(* PLC project SafeLOGIC-1, BrAutomation SafeDESIGNER  4.1.3.320 *)
(* stored: companyURL http://www.br-automation.com, creationDateTime Thu May 07 13:59:02 2020 *)

PROGRAM Zone
  VAR  (* added by the conversion: wires and edge detectors of the diagram *)
    _SAFEBOOL_TO_BOOL91_OUT : BOOL;
    _BOOL_TO_SAFEBOOL159_OUT : SAFEBOOL;
  END_VAR

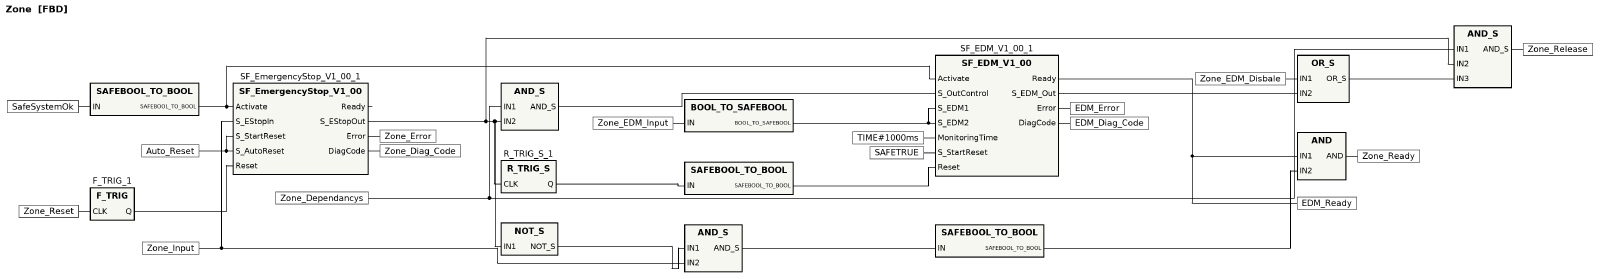
(* FBD diagram, written out as Structured Text *)
_SAFEBOOL_TO_BOOL91_OUT := SAFEBOOL_TO_BOOL(SafeSystemOk);
F_TRIG_1(CLK := Zone_Reset);
SF_EmergencyStop_V1_00_1(Activate := _SAFEBOOL_TO_BOOL91_OUT, S_EStopIn := Zone_Input, S_StartReset := Auto_Reset, S_AutoReset := Auto_Reset, Reset := F_TRIG_1.Q);
_BOOL_TO_SAFEBOOL159_OUT := BOOL_TO_SAFEBOOL(Zone_EDM_Input);
R_TRIG_S_1(CLK := SF_EmergencyStop_V1_00_1.S_EStopOut);
SF_EDM_V1_00_1(Activate := _SAFEBOOL_TO_BOOL91_OUT, S_OutControl := AND_S(Zone_Dependancys, SF_EmergencyStop_V1_00_1.S_EStopOut), S_EDM1 := _BOOL_TO_SAFEBOOL159_OUT, S_EDM2 := _BOOL_TO_SAFEBOOL159_OUT, MonitoringTime := TIME#1000ms, S_StartReset := SAFETRUE, Reset := SAFEBOOL_TO_BOOL(R_TRIG_S_1.Q));
Zone_Release := AND_S(Zone_Dependancys, SF_EmergencyStop_V1_00_1.S_EStopOut, OR_S(Zone_EDM_Disbale, SF_EDM_V1_00_1.S_EDM_Out));
EDM_Error := SF_EDM_V1_00_1.Error;
EDM_Diag_Code := SF_EDM_V1_00_1.DiagCode;
EDM_Ready := SF_EDM_V1_00_1.Ready;
Zone_Ready := SF_EDM_V1_00_1.Ready AND SAFEBOOL_TO_BOOL(AND_S(Zone_Input, NOT_S(SF_EmergencyStop_V1_00_1.S_EStopOut)));
Zone_Diag_Code := SF_EmergencyStop_V1_00_1.DiagCode;
Zone_Error := SF_EmergencyStop_V1_00_1.Error;
END_PROGRAM
